// CODESYS_SoftMotion_Win_V3/Application/Visualizations/JogVis
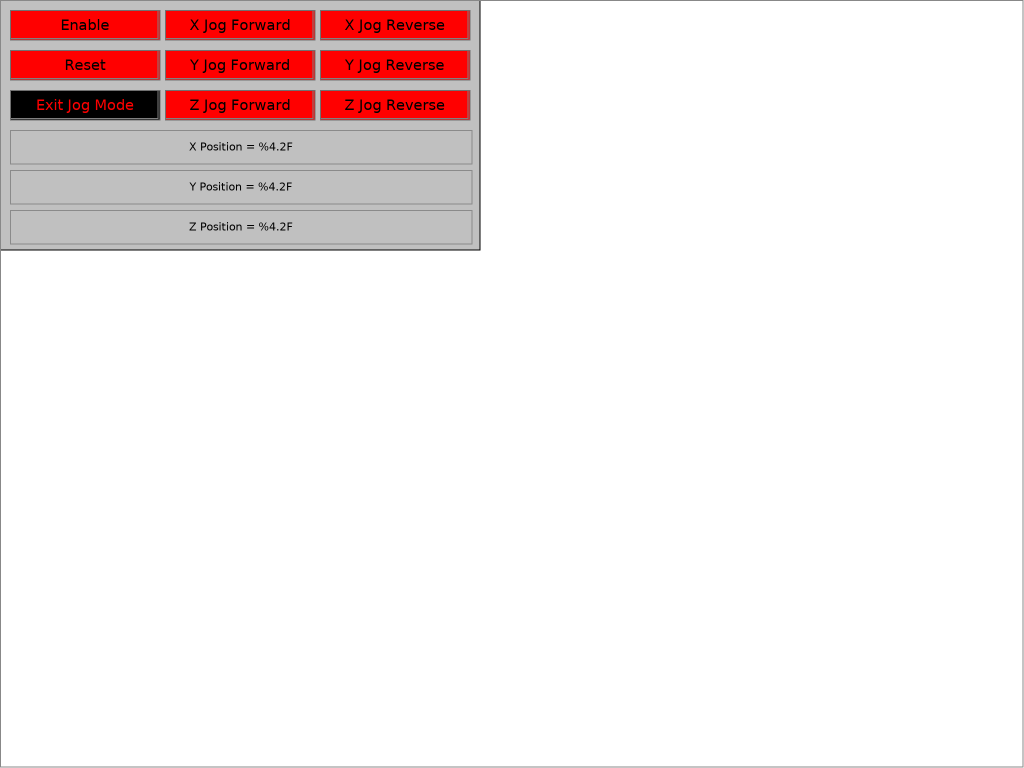
VISUALIZATION JogVis  // 1024x768
    Group (0,0 550x300)
        Rectangle (0,0 480x250)
        Button (10,10 150x30), "Enable"
            OnMouseClick:  ToggleVariable=systemEnable
        Button (165,10 150x30), "X Jog Forward"
            tap JogLogic.xJogFwdPressed
        Button (320,10 150x30), "X Jog Reverse"
            tap JogLogic.xJogRevPressed
        Button (165,50 150x30), "Y Jog Forward"
            tap JogLogic.yJogFwdPressed
        Button (320,50 150x30), "Y Jog Reverse"
            tap JogLogic.yJogRevPressed
        Button (10,50 150x30), "Reset"
            OnMouseClick: execute { JogMotor.systemReset := TRUE; }
        Button (165,90 150x30), "Z Jog Forward"
            tap JogLogic.zJogFwdPressed
        Button (320,90 150x30), "Z Jog Reverse"
            tap JogLogic.zJogRevPressed
        Frame (10,130 462x34), "X Position = %4.2F", text variable: X.fActPosition
            shows SM3_Basic.LinDrive(m_Input_AXISREF := X)
        Frame (10,170 462x34), "Y Position = %4.2F", text variable: Y.fActPosition
            shows SM3_Basic.LinDrive(m_Input_AXISREF := Y)
        Frame (10,210 462x34), "Z Position = %4.2F", text variable: Z.fActPosition
            shows SM3_Basic.LinDrive(m_Input_AXISREF := Z)
        Button (10,90 150x30), "Exit Jog Mode"
            OnMouseClick:  Dialog=JogVis, Result=OK, NumpadKeypadSet=True
END_VISUALIZATION

// CODESYS_SoftMotion_Win_V3/Application/Visualizations/HowToPlay
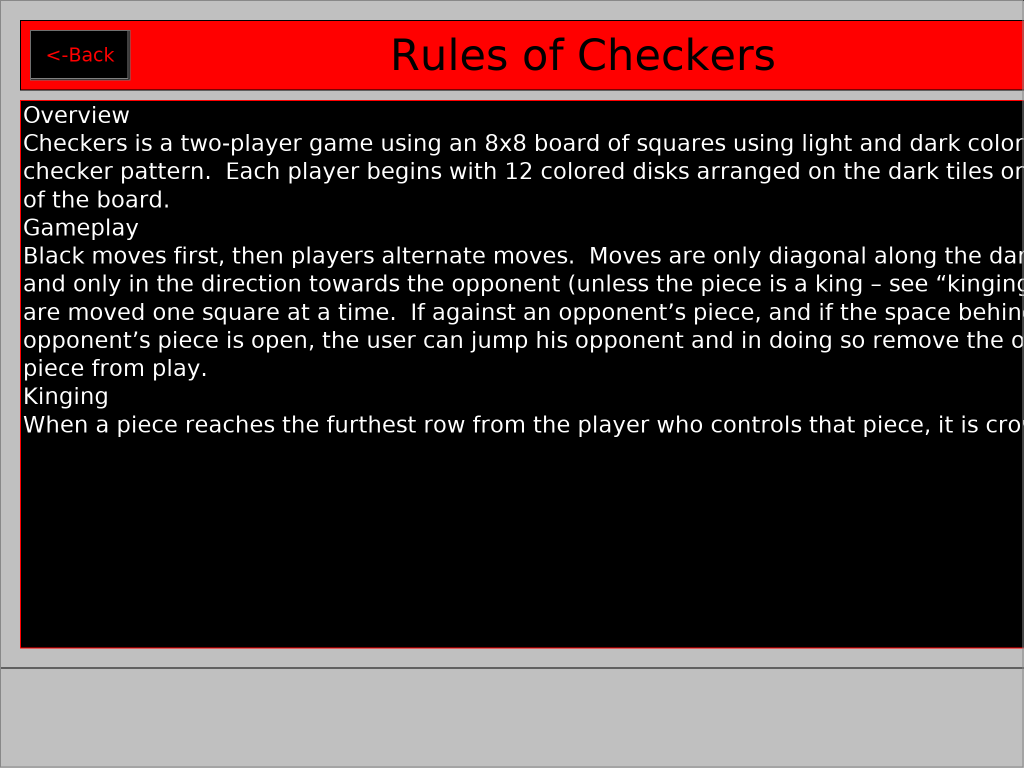
VISUALIZATION HowToPlay  // 1024x768
    Rectangle (0,0 1166x668)
    Textfield (20,100 1126x548), "Overview Checkers is a two-player game using an 8x8 board of squares using light and dark colors in a checker pattern. Each player begins with 12 colored disks arranged on the dark tiles on their side of the board. Gameplay Black moves first, then players alternate moves. Moves are only diagonal along the dark squares and only in the direction towards the opponent (unless the piece is a king – see “kinging”). Pieces are moved one square at a time. If against an opponent’s piece, and if the space behind the opponent’s piece is open, the user can jump his opponent and in doing so remove the opponent piece from play. Kinging When a piece reaches the furthest row from the player who controls that piece, it is crowned and becomes a king. One of the pieces which had been captured is placed on top of the king so that it is twice as high as a single piece. Kings may move both forward and backwards Winning A player wins the game when the opponent cannot make a move. In most cases, this is because all of the opponent's pieces have been captured, but it could also be because all of his pieces are blocked in."
    Textfield (20,20 1126x70), "Rules of Checkers"
    Button (30,30 100x50), "<-Back"
        OnMouseClick:  Dialog=HowToPlay, Result=OK, NumpadKeypadSet=True
END_VISUALIZATION

// CODESYS_SoftMotion_Win_V3/Application/Visualizations/ErrorsCleared
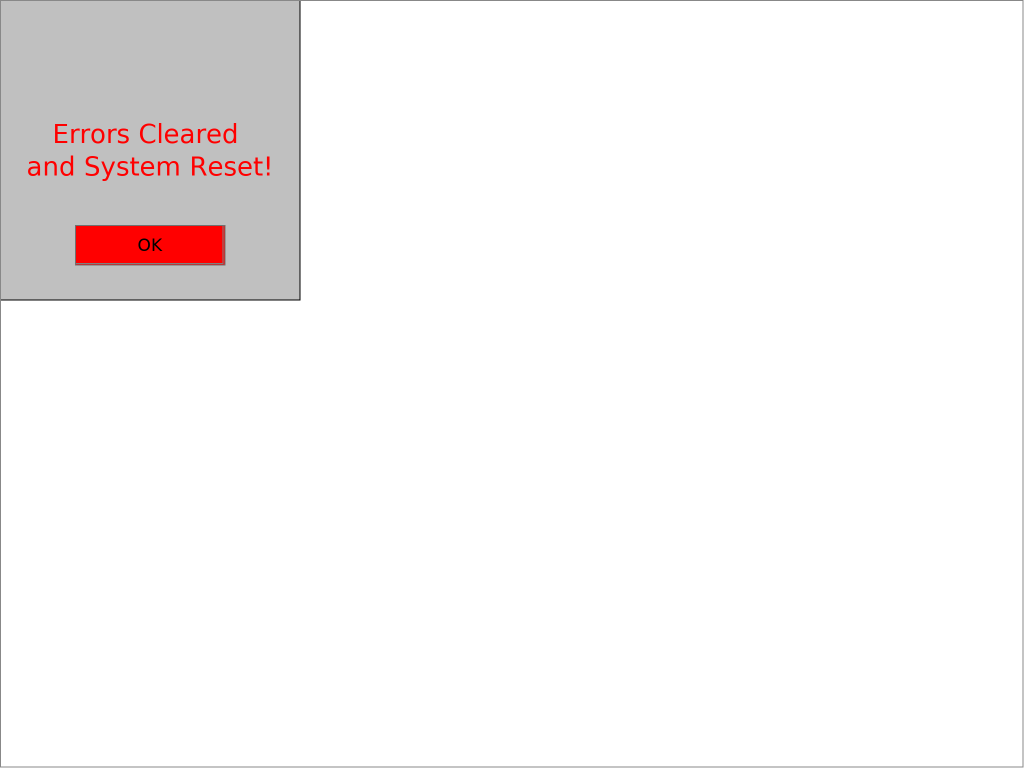
VISUALIZATION ErrorsCleared  // 1024x768
    Rectangle (0,0 300x300), "Errors Cleared and System Reset!"
    Button (75,225 150x40), "OK"
        OnMouseClick:  Dialog=ErrorsCleared, Result=OK, NumpadKeypadSet=True
END_VISUALIZATION

// CODESYS_SoftMotion_Win_V3/Application/Visualizations/Congratulations
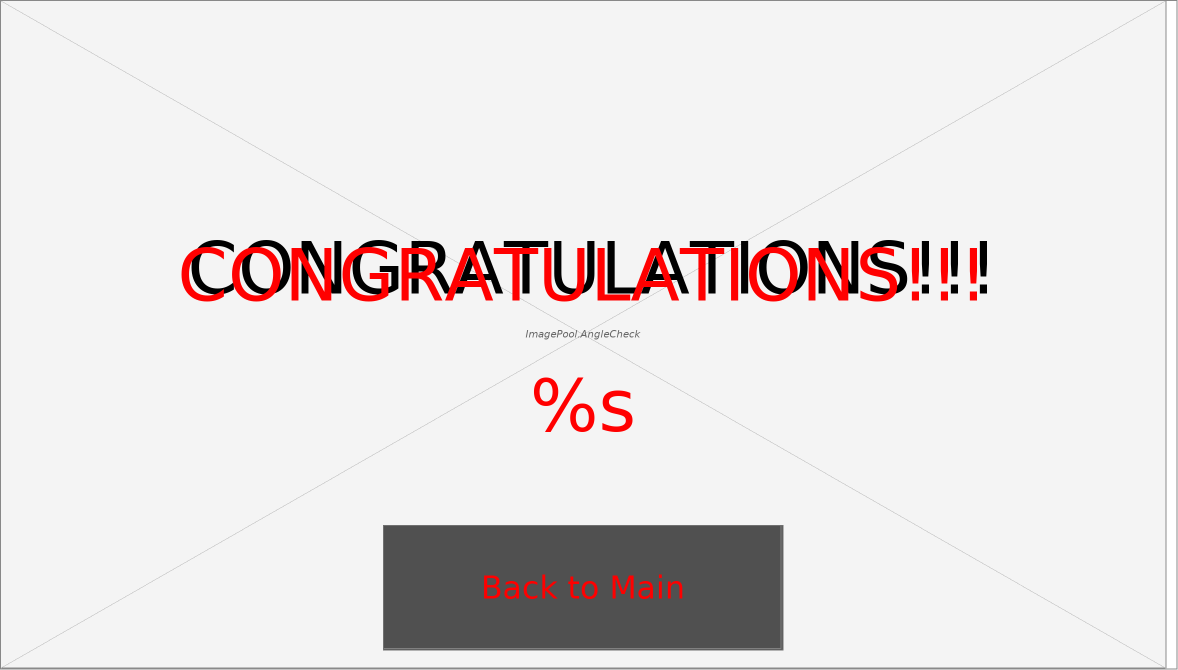
VISUALIZATION Congratulations  // 1178x670
    Image (0,0 1166x668), image: ImagePool.AngleCheck
    Rectangle (10,-7 1166x550), "CONGRATULATIONS!!!"
    Rectangle (0,0 1166x550), "CONGRATULATIONS!!!"
    Button (383,525 400x125), "Back to Main"
    Textfield (0,350 1166x111), "%s", text variable: winnerName
END_VISUALIZATION

(* text COWBELL_PROGRAMMING_STANDARD
*** General Team Guidelines ***

Program Names (Func, FB, Prog): ProgramName, Program_Name
-Which ever way appears more readable

Variable Names: var1, xVelocity, yVel1
-If global axis variable, axis identifier leads descriptive name.  start lowercase, camelCase

Functions, FunctionBlocks: These should not use global variables, if it can be avoided.  
These types should be able to copy and paste into a new program.

( * Header Comment * ) - good for describing chuncks of code
// In line comment - good for describing a single line

Programs, GlobalVars, etc. will be placed in the POUs so that we can work with the simulator from home.  Don't forget to copy programs to the required task!


Functions can only be called, take inputs and have defined outputs.  Good for math or modifiers.
Function Blocks must be called in a program and do not have explicitly defined inputs and outputs.  Good for repetive chunks of code.  
Programs are the only items that are run in the Task Configuration list.  Programs will call Functions and Function Blocks as required.  

*For Visual Stuff, let's try to stay with the Arial family of Fonts
*)

(* text GameInformation
Logins:

Admin : 1234
Tech : 123
User: play
*)
